TYPE HydraulicsPumpsStates :
(
	STOPPED := 0,
	POWERING_ON := 1,
	RESETTING_DRIVES := 2,
	COMMANDING_SAFETY := 3,
	BUILDING_UP_PRESSURE := 4,
	RUNNING := 5,
	STOPPING := 6,
	POWERING_OFF := 7,
	MANUAL := 8,
	ERROR := 9
);
END_TYPE

(* stored: Version 1.1.0.1, ProductVersion 3.1.4019.2
   DUT HydraulicsPumpsStates: Id {9bfdcb81-8441-406e-a13f-42f419c12ec5} *)
